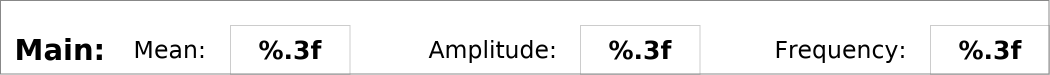
VISUALIZATION VISU_Sine_1  // 1050x75
    Textfield (230,25 120x50), "%.3f", text variable: G_Parameter.fMain_Mean
        OnMouseClick: write the text variable via InputWithLimits, min 0.1, max 0.7
    Textfield (110,25 120x50), "Mean:"
    Textfield (580,25 120x50), "%.3f", text variable: G_Parameter.fMain_Amplitude
        OnMouseClick: write the text variable via InputWithLimits, max 0.2
    Textfield (416,25 154x50), "Amplitude:"
    Textfield (930,25 120x50), "%.3f", text variable: G_Parameter.fMain_Frequency
        OnMouseClick: write the text variable via Edit
    Textfield (761,25 159x50), "Frequency:"
    Textfield (0,25 120x50), "Main:"
END_VISUALIZATION

(* stored: Version 1.1.0.1
   Visu VISU_Sine_1: Id {f8ac259f-06c7-4f75-ad8a-3571cb9713a2} *)
